TYPE STMTargetVelocity :
STRUCT
	velocity : INT;
	acceleration : UINT;
	deceleration : UINT;
END_STRUCT
END_TYPE

(* stored: Version 1.1.0.1, ProductVersion 3.1.4024.9
   DUT STMTargetVelocity: Id {e7a31b1d-ab54-44c5-b0f7-b506d2e0010d} *)
